// TIA Portal V18 export
DATA_BLOCK "ST10_SafetyGate_InterfaceDB"   // DB1140
{ S7_Optimized_Access := 'TRUE' }
// stored: AutoNumber false, MemoryReserve 100
   VAR
      aDev { S7_SetPoint := 'True'} : Array[1..20] of "SafetyGateUDT";
      SafetyDoorLamp { S7_SetPoint := 'True'} : Array[1..20] of Bool;
      H : Struct
         Status_1 : Int;
         Status_2 : Int;
         Status_3 : Int;
         p : Array[0..20] of Bool;
      END_STRUCT;
      J : Struct
         Status_1 : Int;
         Status_2 : Int;
         Status_3 : Int;
         p : Array[0..20] of Bool;
      END_STRUCT;
      K : Struct
         Status_1 : Int;
         Status_2 : Int;
         Status_3 : Int;
         p : Array[0..20] of Bool;
      END_STRUCT;
      L : Struct
         Status_1 : Int;
         Status_2 : Int;
         Status_3 : Int;
         p : Array[0..20] of Bool;
      END_STRUCT;
   END_VAR
BEGIN
END_DATA_BLOCK
